{attribute 'linkalways'} 
{attribute 'no_explicit_call' := 'This FB is a CLASS and must be accessed using methods or properties'}
{attribute 'enable_dynamic_creation'}
FUNCTION_BLOCK Node_F_VN_GetPixel EXTENDS VisionNode
VAR
    ipSrcImage : _ITcVnImage;
    aValue : _TcVnVector4_LREAL;
    nX : _UDINT(0);
    nY : _UDINT(0);
    hrPrev : _HRESULT(S_OK);
	hresult : _HRESULT(S_OK);
END_VAR

METHOD PUBLIC  Clone : I_Node
VAR
	pNode : POINTER TO Node_F_VN_GetPixel;
END_VAR
pNode := __NEW(Node_F_VN_GetPixel);
Clone := pNode^;
END_METHOD

METHOD FB_init : BOOL
VAR_INPUT
	bInitRetains : BOOL; // if TRUE, the retain variables are initialized (warm start / cold start)
	bInCopyCode : BOOL;  // if TRUE, the instance afterwards gets moved into the copy code (online change)
END_VAR
AddInput('ipSrcImage', ipSrcImage);
AddParameter('nX', nX);
AddParameter('nY', nY);
AddInput('hrPrev', hrPrev);
AddOutput('aValue', aValue);
AddOutput('hresult',hresult);
END_METHOD

METHOD PROTECTED  OnExecute : HRESULT
hresult.Value := F_VN_GetPixel(
    ipSrcImage := ipSrcImage.Value,
    aValue := aValue.Value,
    nX := nX.Value,
    nY := nY.Value,
	hrPrev:= hrPrev.Value);
END_METHOD

METHOD PUBLIC PreExecutionCheck
VAR_INPUT
	Check : I_PreExecutionChecks;
END_VAR
Check.IsTrue(ipSrcImage.IsValid, 'ipSrcImage must contain an image');
END_METHOD

END_FUNCTION_BLOCK

(* stored: Version 1.1.0.1, ProductVersion 3.1.4024.13
   POU Node_F_VN_GetPixel: Id {44f30818-257c-01ce-3047-2fb1cae78e0c}, SpecialFunc None
   Folder Constructor: Id {0417244e-bfe4-0ea9-0369-74016f58c6c5}
   Method Clone: Id {ecbe5e94-567f-04d3-1fc7-e32406706d07}
   Method FB_init: Id {72be28f4-23eb-0d85-1abd-0a7efbf41cd8}
   Method OnExecute: Id {59f144fd-6bab-074b-170a-a36533e875fa}
   Method PreExecutionCheck: Id {02a64b13-c74b-0ee4-0bca-2a07e2d7e09b} *)
